Fanuc KAREL source: ko00017.KL

-- PROVISIONAL review KL for V940-1; original PC SHA256 19e0132a617a247b23fc085bbe155e159e05f66ee0d268c3f8c14b3c59501ae4
-- Incomplete behavior may be omitted. Consult companion uncertainty JSON. Do not deploy.
PROGRAM KO00017
%NOLOCKGROUP
-- UNRESOLVED_DECL P1 type=000106
-- UNRESOLVED_DECL P2 type=000106
-- UNRESOLVED_DECL P3 type=000106
-- UNRESOLVED_DECL OUT type=000101
BEGIN
  -- V9_ZERO_TABLE_METADATA_HINT layout=0001; no indexed target words; source/name/runtime held
  -- UNRESOLVED_PC offsets 5-65; opcodes 27,27,49,7E,AD,27,49,7E,AD,27,49,7E,AD,76,7E,4A
  -- UNRESOLVED_PC offsets 70-74; opcodes 7F
END KO00017
